FUNCTION_BLOCK ConvCtrl (* Basic Function Block Type *)
  (* Standard: 61499-2 *)
  (* Version 0.0, 3/23/2016, Aalto_IT, nxtControl GmbH, Template *)
  PACKAGE Main;
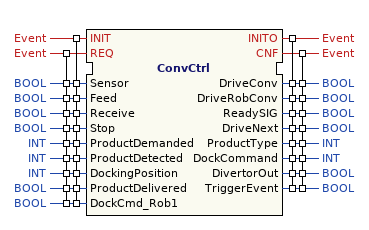
  EVENT_INPUT
    INIT WITH Sensor, Feed, Receive, Stop, ProductDemanded, ProductDetected, DockingPosition, ProductDelivered, DockCmd_Rob1; (* Initialization Request *)
    REQ WITH Sensor, Feed, Receive, Stop, ProductDemanded, ProductDetected, DockingPosition, ProductDelivered, DockCmd_Rob1; (* Normal Execution Request *)
  END_EVENT
  EVENT_OUTPUT
    INITO WITH DriveConv, DriveRobConv, ReadySIG, DriveNext, ProductType, DockCommand, DivertorOut, TriggerEvent; (* Initialization Confirm *)
    CNF WITH DriveConv, DriveRobConv, ReadySIG, DriveNext, ProductType, DockCommand, DivertorOut, TriggerEvent; (* Execution Confirmation *)
  END_EVENT
  VAR_INPUT
    Sensor : BOOL;
    Feed : BOOL; (* Input event qualifier *)
    Receive : BOOL;
    Stop : BOOL;
    ProductDemanded : INT;
    ProductDetected : INT;
    DockingPosition : INT;
    ProductDelivered : BOOL;
    DockCmd_Rob1 : BOOL;
  END_VAR
  VAR_OUTPUT
    DriveConv : BOOL; (* Output event qualifier *)
    DriveRobConv : BOOL;
    ReadySIG : BOOL;
    DriveNext : BOOL;
    ProductType : INT;
    DockCommand : INT;
    DivertorOut : BOOL;
    TriggerEvent : BOOL;
  END_VAR
  VAR
    TimeStamp : DATE_AND_TIME;
  END_VAR
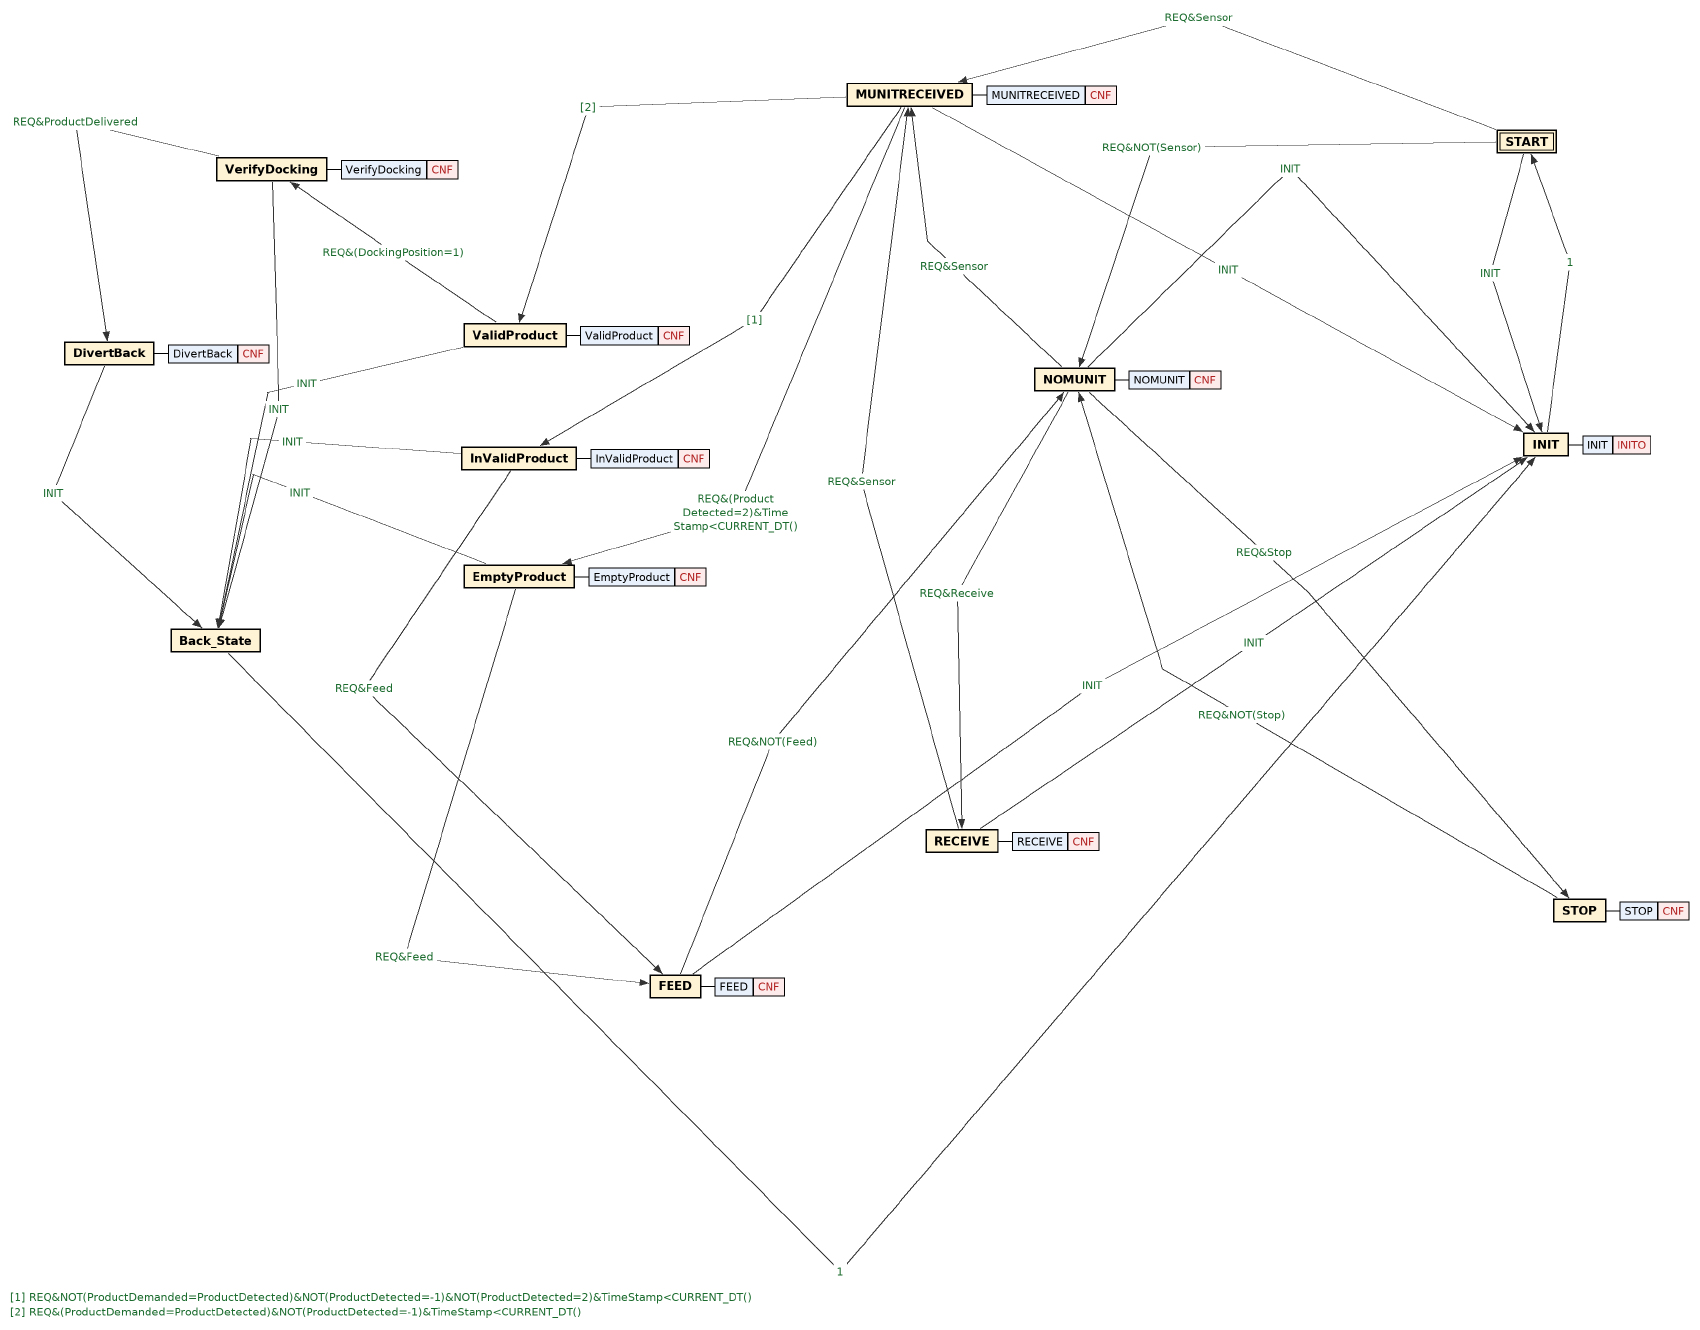
  EC_STATES
    START; (* Initial State *)
    INIT : INIT -> INITO; (* Initialization *)
    FEED : FEED -> CNF; (* Normal execution *)
    MUNITRECEIVED : MUNITRECEIVED -> CNF; (* Normal execution *)
    NOMUNIT : NOMUNIT -> CNF;
    RECEIVE : RECEIVE -> CNF;
    STOP : STOP -> CNF;
    ValidProduct : ValidProduct -> CNF;
    InValidProduct : InValidProduct -> CNF;
    EmptyProduct : EmptyProduct -> CNF;
    Back_State;
    VerifyDocking : VerifyDocking -> CNF;
    DivertBack : DivertBack -> CNF;
  END_STATES
  EC_TRANSITIONS
    START TO INIT := INIT;
    INIT TO START := 1;
    NOMUNIT TO MUNITRECEIVED := REQ&Sensor;
    FEED TO NOMUNIT := REQ&NOT(Feed);
    RECEIVE TO MUNITRECEIVED := REQ&Sensor;
    START TO MUNITRECEIVED := REQ&Sensor;
    NOMUNIT TO RECEIVE := REQ&Receive;
    START TO NOMUNIT := REQ&NOT(Sensor);
    RECEIVE TO INIT := INIT;
    NOMUNIT TO INIT := INIT;
    FEED TO INIT := INIT;
    MUNITRECEIVED TO INIT := INIT;
    NOMUNIT TO STOP := REQ&Stop;
    STOP TO NOMUNIT := REQ&NOT(Stop);
    MUNITRECEIVED TO ValidProduct := REQ&(ProductDemanded=ProductDetected)&NOT(ProductDetected=-1)&TimeStamp<CURRENT_DT();
    MUNITRECEIVED TO InValidProduct := REQ&NOT(ProductDemanded=ProductDetected)&NOT(ProductDetected=-1)&NOT(ProductDetected=2)&TimeStamp<CURRENT_DT();
    MUNITRECEIVED TO EmptyProduct := REQ&(ProductDetected=2)&TimeStamp<CURRENT_DT();
    InValidProduct TO Back_State := INIT;
    EmptyProduct TO Back_State := INIT;
    InValidProduct TO FEED := REQ&Feed;
    EmptyProduct TO FEED := REQ&Feed;
    Back_State TO INIT := 1;
    ValidProduct TO VerifyDocking := REQ&(DockingPosition=1);
    VerifyDocking TO Back_State := INIT;
    ValidProduct TO Back_State := INIT;
    VerifyDocking TO DivertBack := REQ&ProductDelivered;
    DivertBack TO Back_State := INIT;
  END_TRANSITIONS
  ALGORITHM INIT IN ST: (* Initialization algorithm *)
;
DriveConv:=0;
ReadySIG:=1;
DriveNext:=0;
ProductDetected := -1;
ProductType := -1; // Garbage\
DivertorOut := 0;
DriveRobConv := FALSE;
TriggerEvent := FALSE;
  END_ALGORITHM
  ALGORITHM FEED IN ST:
DriveConv:=1;
ReadySIG:=0;
DriveNext := 1;
DivertorOut := 0;
DriveRobConv := FALSE;
TriggerEvent := FALSE;
  END_ALGORITHM
  ALGORITHM MUNITRECEIVED IN ST:
// stop the Conveyor and do color detection.
DriveConv:=0; //stop the Conveyor
ReadySIG:=0;
DriveNext:=0;
TimeStamp:=ADD_DT_TIME(CURRENT_DT(),T#5.0s);
DivertorOut := 0;
DriveRobConv := FALSE;
TriggerEvent := FALSE;
  END_ALGORITHM
  ALGORITHM NOMUNIT IN ST:
// Drive the Conveyor Initially Regardless of the Value of the Sensor.
DriveConv:=1;
ReadySIG:=1;
DriveNext:=0;
//ProductDetected := -1;
//ProductType := -1; // Garbage
DivertorOut := 0;
DriveRobConv := FALSE;
TriggerEvent := FALSE;
  END_ALGORITHM
  ALGORITHM RECEIVE IN ST:
DriveConv:=1;
ReadySIG:=1;
DriveNext:=0;
DivertorOut := 0;
DriveRobConv := FALSE;
TriggerEvent := FALSE;
  END_ALGORITHM
  ALGORITHM STOP IN ST:
DriveConv:=0;
ReadySIG:=0;
DriveNext:=0;
DivertorOut := 0;
DriveRobConv := FALSE;
TriggerEvent := FALSE;
  END_ALGORITHM
  ALGORITHM ValidProduct IN ST:
;
// Product is Valid, just drive the conveyor and Open Up the Divertor.
DriveConv:= 0; //stop the Conveyor
ReadySIG:=0;
DriveNext:=0;
ProductType := 1; // Valid Product
DivertorOut := 0;
DriveRobConv := FALSE;
DockCommand := 1;
TriggerEvent := TRUE;
  END_ALGORITHM
  ALGORITHM InValidProduct IN ST:
;
// Product is In-Valid, and we need Jack1 to remove the WP.
DriveConv:=1; //stop the Conveyor
ReadySIG:=0;
DriveNext:=0; // Should It be 1 ?????
ProductType := 0; // In-Valid Product
DivertorOut := 0;
DriveRobConv := FALSE;
TriggerEvent := FALSE;
  END_ALGORITHM
  ALGORITHM EmptyProduct IN ST:
;
// Product is Empty, Jack2 will fill it up !
DriveConv := 1; //stop the Conveyor
ReadySIG:=0;
DriveNext:=0;
ProductType := 2; // Empty Product
DivertorOut := 0;
DriveRobConv := FALSE;
TriggerEvent := FALSE;
  END_ALGORITHM
  ALGORITHM VerifyDocking IN ST:
;
// Robotino has docked.
DriveConv:=1; //stop the Conveyor
ReadySIG:=0;
DriveNext:=0;
ProductType := 1; // Valid Product
DivertorOut := 1;// Make the Output for NxtHigh here...
DriveRobConv := TRUE;
TriggerEvent := FALSE;
  END_ALGORITHM
  ALGORITHM DivertBack IN ST:
;
// product has reached final station. Put the DivertorBack.
DriveConv:=1; //stop the Conveyor
ReadySIG:=0;
DriveNext:=0;
ProductType := 1; // Valid Product
DivertorOut := 0;
DriveRobConv := FALSE;
TriggerEvent := FALSE;
  END_ALGORITHM
END_FUNCTION_BLOCK
